# EPICS substitutions: src/iocdoc/testfiles/iocBoot/ioc495idc/templates/xradia_seamless_motion.substitutions
# $File: //ASP/Dev/SBS/3_Beamlines/3_09_SR05ID01_XFM/3_09_4_Controls/3_09_4_2_Equipment_Control/Xradia/Xradia_Seamless_MotionApp/Db/xradia_seamless_motion.substitutions $
# $Revision: #2 $
# $DateTime: 2009/09/15 18:34:32 $
# Last checked in by: $Author: starritt $
#
# Description:
# Creates records to extract the piezo X/Y voltages and relative positions,
# and also to control hybrid, i.e. seamless, motion.
#
#
# Copyright (c) 2009 Australian Synchrotron
#
# This library is free software; you can redistribute it and/or
# modify it under the terms of the GNU Lesser General Public
# Licence as published by the Free Software Foundation; either
# version 2.1 of the Licence, or (at your option) any later version.
#
# This library is distributed in the hope that it will be useful,
# but WITHOUT ANY WARRANTY; without even the implied warranty of
# MERCHANTABILITY or FITNESS FOR A PARTICULAR PURPOSE.  See the GNU
# Lesser General Public Licence for more details.
#
# You should have received a copy of the GNU Lesser General Public
# Licence along with this library; if not, write to the Free Software
# Foundation, Inc., 51 Franklin St, Fifth Floor, Boston, MA 02110-1301 USA.
#
# Contact details:
# andrew.starritt@synchrotron.org.au
# 800 Blackburn Road, Clayton, Victoria 3168, Australia.
#
# Modications:
# Argonne National Laboratory
# Advance Photon Source (APS)
# APS Engineering Support (AES) Division
# Beamline Controls and Data Acquisition (BCDA) Group
# David M. Kline [ dkline@aps.anl.gov ]
#

file "$(TOP)/495idcApp/Db/xradia_seamless_motion.db"
{
pattern
{P               PORT        XY      VVAR        MINRP       MAXRP       LIMIT   OFFSET  STOP    PIEZO       FOM}

{"495idcnpi:",   "pmac2E",   "X",    "M102",     "-6.8",     "+6.8",     "2.8",  "10.0", "#2k", "$(P)m34",  "$(P)m10"}
{"495idcnpi:",   "pmac2E",   "Y",    "M202",     "-2.27",    "+2.27",    "1.12", "2.0",  "#3k", "$(P)m35",  "$(P)m11"}

}

# end
